(* IEC 61131-3 sources: plc_generation_empirical_study/datasets/packages/internal_v0_1/qualification_only/C05_M01_off_delay_fan, 1 file *)

(* ---- reference.st ---- *)
FUNCTION_BLOCK C05_M01_off_delay_fan
VAR_INPUT
    Demand : BOOL;
    SafetyTrip : BOOL;
END_VAR
VAR_OUTPUT
    Fan : BOOL;
    RunOn : BOOL;
END_VAR
VAR
    OffTimer : TOF;
END_VAR

OffTimer(IN := Demand AND (NOT SafetyTrip), PT := T#300ms);
IF SafetyTrip THEN
    Fan := FALSE;
ELSE
    Fan := OffTimer.Q;
END_IF;
RunOn := (NOT Demand) AND Fan;

END_FUNCTION_BLOCK
